TYPE ST_Position :
STRUCT
	// @1:X
	x	:	LREAL;
	// @1:Y
	y	: 	LREAL;
	// @1:Z	
	Z	: 	LREAL;
END_STRUCT
END_TYPE

(* stored: Version 1.1.0.1, ProductVersion 3.1.4022.6
   DUT ST_Position: Id {54512147-6c2e-4106-bc2c-b21f46de2f63} *)
